{attribute addProperty BoxType "EL9550-0010-0016"}
{attribute addProperty Id "Status_UpAT %I*Status_Up_B12359DC1620Status_UsAT %I*Status_Us_B12359DC1620WcStateAT %I*WcState_98A4DF7520.250InfoDataAT %I*InfoData_192954DE1620"}
{attribute addProperty CRC "3568038920"}
{attribute addProperty SizeInBites "50"}
{attribute addProperty SizeInBytes "6.25"}
TYPE EL9550_B50CDD11 :
STRUCT
	{attribute addProperty Name "Status_Up"}
	Status_Up : Status_Up_B12359DC;
	{attribute addProperty Name "Status_Us"}
	Status_Us : Status_Us_B12359DC;
	{attribute addProperty Name "WcState"}
	WcState : WcState_98A4DF75;
	{attribute addProperty Name "InfoData"}
	InfoData : InfoData_192954DE;
END_STRUCT
END_TYPE

(* stored: Version 1.2.0.0, ProductVersion 3.1.4024.9
   DUT EL9550_B50CDD11: Id {fa68be54-a7a0-4cc6-8486-e13553db23f9} *)
